{attribute addProperty BoxType "AT2050-0500-0019"}
{attribute addProperty Id "A_0094_AT2021_5250_0018_AT2021_5250AT2021_C5E5984862678.25"}
{attribute addProperty CRC "3875018064"}
{attribute addProperty SizeInBites "626"}
{attribute addProperty SizeInBytes "78.25"}
TYPE A_0050_AT2050_0500_0019_E6F81550 EXTENDS AT2050_BA5A9548 :
STRUCT
	{attribute addProperty Name "A_0094_AT2021_5250_0018_AT2021_5250"}
	A_0094_AT2021_5250_0018_AT2021_5250 : AT2021_C5E59848;
END_STRUCT
END_TYPE

(* stored: Version 1.2.0.0, ProductVersion 3.1.4024.9
   DUT A_0050_AT2050_0500_0019_E6F81550: Id {28959489-1f30-473f-80d7-f81e90b6f7c7} *)
